// TwinCAT 3 PLC project BaseElementsSample
// ProgramVersion: 3.1.4020.1
// libraries:
//   Base_Elements,0.0.1.68,Vistaprint
//   Base_PLC,0.3.6.2,Vistaprint
//   Tc2_EtherCAT,3.3.7.0,Beckhoff Automation GmbH
//   Tc2_SerialCom,3.3.5.0,Beckhoff Automation GmbH
//   Tc2_Standard,3.3.1.0,Beckhoff Automation GmbH
//   Tc2_System,3.4.13.0,Beckhoff Automation GmbH
//   Tc2_TcpIp,3.3.3.0,Beckhoff Automation GmbH
//   Tc2_Utilities,3.3.14.0,Beckhoff Automation GmbH
//   Tc3_Interfaces,3.4.2.0,Beckhoff Automation GmbH
//   Tc3_MemMan,3.3.1.0,Beckhoff Automation GmbH
//   Tc3_Module,3.3.11.0,Beckhoff Automation GmbH
// project tree:
//   DUTs/ E_CtrlId.TcDUT, T_HashInfo.TcDUT (not stored)
//   DUTs/GVLs/ Global.TcGVL, Io.TcGVL
//   POUs/Program/ MiddlePRG_1.TcPOU, SlowPRG_1.TcPOU (not stored), FastPRG_1.TcPOU
//   / Task_Fast.TcTTO, Task_Middle.TcTTO (not stored), Task_Slow.TcTTO (not stored)
// (motion and I/O tree: see PLC project base_elements)
// real-time tasks:
//   TASK Task_Fast: cycle T#2ms, priority 4, ADS port 350
//   TASK Task_Slow: cycle T#50000us, priority 8, ADS port 351
//   TASK Task_Middle: cycle T#10ms, priority 6, ADS port 352

CONFIGURATION BaseElementsSample
    RESOURCE PLC ON TwinCAT3
        TASK Task_Fast(INTERVAL := T#2ms, PRIORITY := 4);
        PROGRAM FastPRG_1 WITH Task_Fast : FastPRG_1;
    END_RESOURCE
END_CONFIGURATION

// ---- DUTs/E_CtrlId.TcDUT
TYPE E_CtrlId :
(
	//not defined after startup...
	NONE,
	RFW_11,
	CYL_1,
	VPC_1,	
	UMC_1,	
	PRS_1,	
	BCC_1,
	DRV_1,
	RFW_12,
	ACL_1,
	VLV_1,
	ECD_1,
	E_CtrlIdMax
);
END_TYPE

// ---- DUTs/GVLs/Global.TcGVL
VAR_GLOBAL
	/// instance array of all controller instances
	g_a_pCtrlInst: ARRAY[0..E_CtrlId.E_CtrlIdMax] OF POINTER TO fb_CtrlBase;
	/// common interface array of all controllers (main use for PLC)
	g_a_pCtrlCIf: ARRAY[0..E_CtrlId.E_CtrlIdMax] OF POINTER TO T_Ctrl_CIf;
	
	/// global alarm manager
	g_p_fbAlm_Man: POINTER TO FB_Alm_Man;
	
	///Global accesss of driver init in faster cycles
	g_pFB_RFR: POINTER TO FB_RFR;	
	g_pFB_BCD: POINTER TO FB_BCD;
	g_pFB_RFD: POINTER TO FB_RFD;
	
	g_uinStartProzess : UINT; // For StartUp order
  	
END_VAR

VAR_GLOBAL CONSTANT
	c_uinCntTaskClass : UINT := 3;	// Count of Task Classes
END_VAR

// ---- DUTs/GVLs/Io.TcGVL
VAR_GLOBAL
	In_bol_11_0_B1_Doublestopper_full AT %I* : BOOL; //VOLLMELDUNG DOPPELSTOPPER
	Out_bol_11_0_Q2_Doublestopper AT %Q* : BOOL; //DOPPELSTOPPER
	In_bol_11_0_B3_Doublestopper_full AT %I* : BOOL; //VOLLMELDUNG DOPPELSTOPPER
	Out_bol_11_0_Q4_Doublestopper AT %Q* : BOOL; //DOPPELSTOPPER
	In_bol_11_0_B5_Seperator_full AT %I* : BOOL; //VOLLMELDUNG VEREINZELUNG
	In_bol_11_0_B6_Hanger_in_Seperator AT %I* : BOOL; //BUEGEL IN VEREINZELUNG
	Out_bol_11_0_Q7_Seperator AT %Q* : BOOL; //VEREINZELUNG
	Out_bol_11_0_Q8_Control_stopper AT %Q* : BOOL; //KONTROLLSTOPPER
	Out_bol_11_0_A1_Drive_On AT %Q* : BOOL; //ANTRIEB EIN
	In_bol_11_0_A1_Motor_Protection AT %I* : BOOL; //MOTORSCHUTZ AUSGELOEST
	In_bol_11_0_B13_Doublestopper_full AT %I* : BOOL; //VOLLMELDUNG DOPPELSTOPPER
	Out_bol_11_0_Q14_Doublestopper AT %Q* : BOOL; //DOPPELSTOPPER
	In_bol_11_0_B15_New_part AT %I* : BOOL; //NEUES TEIL
	In_bol_EmergencyOff AT %I* : BOOL; // Emergency Off Button
	Out_bolLED_RD AT %Q* : BOOL; // Red LED
	Out_bolLED_YE AT %Q* : BOOL; // Yellow LED
	Out_bolLED_GN AT %Q* : BOOL; // Green LED
	Out_bolBeep AT %Q* : BOOL; // Beeper
END_VAR

// ---- POUs/Program/FastPRG_1.TcPOU
PROGRAM FastPRG_1
VAR
	bolPlcStartupDone: BOOL := FALSE;
	bolHostInitDone: BOOL := FALSE;
	bolInitDone: BOOL := FALSE;

	// RFID driver
	fbRFR_11: FB_RFR;
	fbRFD_12: FB_RFD;
	// Barcode driver
	fbBCD_1: FB_BCD;
	
	fbHashTable : FB_GHT;
	uliBarcodeIn	: ULINT := 0;
	uliBarcodeOut	: ULINT := 0;

	rHashInfo	: T_HashInfo;
	pHashInfo	: POINTER TO T_HashInfo;	

END_VAR

(*__________________________________________________________________________________________________
¦	
¦	Vistaprint Schweiz GmbH
¦	CH - 8401 Winterthur
¦
¦	www.vistaprint.ch - info@vistaprint.ch
¦___________________________________________________________________________________________________

Function desription:
call of all controller (FUB) for the fast task class.

for the RFID is necessary to call to driver FUB at about 2-3ms for reaching baudhrate!

History:
Version		Date			Author		Comment
---------------------------------------------------------------------------------------------------
0.00.1		25.09.2013		AVME/KVO	Start history
0.00.2		07.01.2014		AVME/DSC 	Insert barcode driver example
0.00.3		06.01.2014		AVME/PRE	Implement RFW for Promo RFID Reader-Writer
0.00.4		13.01.2014		AVME/PRE	Implement Starup Cycle
___________________________________________________________________________________________________*)

// -----------------------------------------------------------------------------------------------
// Initialize the PLC Parameter and check the PLC health
// -----------------------------------------------------------------------------------------------
IF (NOT bolPlcStartupDone) THEN
	bolPlcStartupDone := TRUE;	
	
	// init	
	g_pFB_RFR := ADR(fbRFR_11);
	g_pFB_RFD := ADR(fbRFD_12);

	g_pFB_BCD := ADR(fbBCD_1);
	g_uinStartProzess:=1; // For StartUp order

	fbHashTable.Initialize();
END_IF
// -----------------------------------------------------------------------------------------------


// -----------------------------------------------------------------------------------------------
// The host system is downloading all parameter at startup. 
// bolPlcStartupDone will be set to true after the Host is done with the initialization
// -----------------------------------------------------------------------------------------------
IF (bolPlcStartupDone AND (NOT bolHostInitDone) AND NOT bolInitDone AND (g_uinStartProzess>=c_uinCntTaskClass)) THEN
	bolHostInitDone := TRUE;
	g_uinStartProzess := 11; // For StartUp order
END_IF
// -----------------------------------------------------------------------------------------------


// -----------------------------------------------------------------------------------------------
// Start PLC code initialization
// -----------------------------------------------------------------------------------------------
IF NOT bolInitDone AND bolPlcStartupDone AND bolHostInitDone AND (g_uinStartProzess>=(10+c_uinCntTaskClass)) THEN
		
	bolInitDone := TRUE;
	g_uinStartProzess := 21; // For StartUp order
END_IF
// -----------------------------------------------------------------------------------------------

// -----------------------------------------------------------------------------------------------
// Normal Run mode after all the initialization is done
// -----------------------------------------------------------------------------------------------
IF (bolInitDone AND bolPlcStartupDone AND bolHostInitDone AND (g_uinStartProzess>=(20+c_uinCntTaskClass))) THEN
	
	//****************************************************************************************************
	// cyclic controller calls
	//****************************************************************************************************
	//fbRFR_11();
	//fbRFD_12();
	fbBCD_1();
	
	IF uliBarcodeIn <> 0 THEN
		pHashInfo := __NEW(T_HashInfo);
		pHashInfo^.strBarcode := ULINT_TO_STRING(uliBarcodeIn);
		fbHashTable.AddItem(uliBarcodeIn, pHashInfo);
		uliBarcodeIn := 0;
	END_IF
	
	IF uliBarcodeOut <> 0 THEN
		pHashInfo := fbHashTable.Lookup(uliBarcodeOut, TRUE);
		MEMCPY(ADR(rHashInfo), pHashInfo, SIZEOF(T_HashInfo));
		__DELETE(pHashInfo);
		uliBarcodeOut := 0;
	END_IF
END_IF
// -----------------------------------------------------------------------------------------------

END_PROGRAM

// ---- POUs/Program/MiddlePRG_1.TcPOU
PROGRAM MiddlePRG_1
VAR
	fbAlm_Man: FB_Alm_Man; // alarm manager
	
	bolPlcStartupDone: BOOL := FALSE;
	bolHostInitDone: BOOL := FALSE;
	bolInitDone: BOOL := FALSE;
	uinTaskNbr : UINT := 2; // MiddleTask is Task Nr 2
	fbRFW_11: FB_RFW;
	fbRFW_12: FB_RFW;
	fbBCC_1: FB_BCC;
	fbCYL_1: FB_CYL;
	fbPRS_1: FB_PRS;
	fbUMC_1: FB_UMC;
	fbVPC_1: FB_VPC;
	fbDRV_1: FB_DRV;
	pTmpSIf_RFW: POINTER TO Base_Elements.T_Ctrl_SIf_RFW;
	pTmpSIf_BCC: POINTER TO T_Ctrl_SIf_BCC;
	fbVLV_1: FB_VLV;
	
	// ADS Client Example
	fbACL_1: FB_ACL;
	sCon01_ShirtStream: T_ADS_ConnectionData; 			// Example: Read connection to shirt stream PLC (Port 851) drive FUB interface .cur
	DrvCurData: T_Ctrl_SIf_DRV_Cur;	
	sCon02_ShirtStream: T_ADS_ConnectionData; 			// Example: Write connection to shirt stream PLC (Port 851) drive FUB interface .par
	DrvParData: T_Ctrl_SIf_DRV_Par;	
	sCon03_ShirtStream: T_ADS_ConnectionData; 			// Example: Write connection to shirt stream PLC (Port 852) drive FUB interface .cfg
	DrvCfgData: T_Ctrl_SIf_DRV_Cfg;	
	// ADS Client Example
	
	// EtherCAT Diagnose
	fbECD_1: FB_ECD;
	pTmpSIf_ECD: POINTER TO T_Ctrl_SIf_ECD;

	fbSGT_1: 		FB_SGT;		// Signal tower	
	pDRV_CIf:		POINTER TO Base_PLC.T_Ctrl_CIf; // Used for Signal tower example
	pDRV_SIf:		POINTER TO Base_Elements.T_Ctrl_SIf_DRV; // Used for Signal tower example
	
	// close all Ethernet sockets
	fbSocketCloseAll : FB_SocketCloseAll;
END_VAR

(*__________________________________________________________________________________________________
¦	
¦	Vistaprint Schweiz GmbH
¦	CH - 8401 Winterthur
¦
¦	www.vistaprint.ch - info@vistaprint.ch
¦___________________________________________________________________________________________________

Function desription:
call of all controller (FUB) for the middle task class.


History:
Version		Date			Author		Comment
---------------------------------------------------------------------------------------------------
0.00.1		25.09.2013		AVME/KVO	Start history
0.00.2		12.11.2013		VP/RE		Local AlarmManager
0.00.3		07.01.2014		AVME/DSC 	Insert barcode reader example
0.00.4		08.01.2014		AVME/MRU	Insert DRV example
0.00.5		06.01.2014		AVME/PRE	Implement RFW for Promo Read and Write RFID Reader
0.00.6		13.01.2014		AVME/PRE	Implement Starting Up Process
0.00.7		05.02.2014		AVME/DSC	Insert ADS client example
0.00.8		06.03.2014		AVME/DSC	Insert FB_VLV example
0.00.9		17.06.2014		AVME/MRU	SGT example added
0.00.10		24.10.2014		HLV/MAH		close all sockets on PLC init

___________________________________________________________________________________________________*)

// -----------------------------------------------------------------------------------------------
// Initialize the PLC Parameter and check the PLC health
// -----------------------------------------------------------------------------------------------
IF (NOT bolPlcStartupDone) AND (g_uinStartProzess>=(uinTaskNbr-1)) THEN
	
	// init	
	// Level0 -------------------------------------------------------------------
	
	// RFID Reader, element Controller in this Task, Driver in fastest Task class
	fbRFW_11.iniAllCtrlArrays(ADR(g_a_pCtrlInst),ADR(g_a_pCtrlCIf),E_CtrlId.RFW_11); // init and entry fb_instance in global fb pointer array
	fbRFW_11.pRFD_SIf := g_pFB_RFR^.getSIf();
	pTmpSIf_RFW := fbRFW_11.getCtrlSIf();
	pTmpSIf_RFW^.Cfg.eTyp := E_Typ_RFW.RF382R;
	// the following parameters are not needed at the moment because the parameters will not be written down for RF382R at the moment
	pTmpSIf_RFW^.Cfg.stNetId := '192.168.2.123.1.1'; //PLC NetId
	pTmpSIf_RFW^.Cfg.uinSlaveAddr := 1024; //Io card Ethercat adress 
	pTmpSIf_RFW^.Cfg.bolGetTrayIDAuto := FALSE;
	
	// RFID Reader, element Controller in this Task, Drive in fastest Task class
	fbRFW_12.iniAllCtrlArrays(ADR(g_a_pCtrlInst),ADR(g_a_pCtrlCIf),E_CtrlId.RFW_12); // init and entry fb_instance in global fb pointer array
	fbRFW_12.pRFD_SIf := g_pFB_RFD^.getSIf();
	pTmpSIf_RFW := fbRFW_12.getCtrlSIf();
	pTmpSIf_RFW^.Cfg.eTyp := E_Typ_RFW.RF310R;
	// the following parameters are not needed at the moment because the parameters will not be written down for RF382R at the moment
	pTmpSIf_RFW^.Cfg.stNetId := '192.168.2.123.1.1'; //PLC NetId
	pTmpSIf_RFW^.Cfg.uinSlaveAddr := 1024; //Io card Ethercat adress 
	pTmpSIf_RFW^.Cfg.bolGetTrayIDAuto := TRUE;
	
	// *********************************************************
	// Barcode reader example
	// *********************************************************
	
	// Barcode reader, element Controller in this Task, Driver in fastest Task class
	fbBCC_1.iniAllCtrlArrays(ADR(g_a_pCtrlInst),ADR(g_a_pCtrlCIf),E_CtrlId.BCC_1); // init and entry fb_instance in global fb pointer array
	fbBCC_1.pBCD_SIf_In := g_pFB_BCD^.getSIf();
	pTmpSIf_BCC := fbBCC_1.getCtrlSIf();
	// configuration	
	pTmpSIf_BCC^.Cfg.strSensorIPAdr := '192.168.70.28';
	pTmpSIf_BCC^.Cfg.udiSensorPort := 2111;
	pTmpSIf_BCC^.Cfg.iSensorType := E_BCD_Type.SICK;
	(*
	pTmpSIf_BCC^.Cfg.strSensorIPAdr := '192.168.1.103';
	pTmpSIf_BCC^.Cfg.udiSensorPort := 9004;
	pTmpSIf_BCC^.Cfg.iSensorType := E_BCD_Type.KEYENCE;
	*)
	// *********************************************************
	// ADS client example
	// *********************************************************
	
	// ADS client connection
	fbACL_1.iniAllCtrlArrays(ADR(g_a_pCtrlInst),ADR(g_a_pCtrlCIf),E_CtrlId.ACL_1); // init and entry fb_instance in global fb pointer array

	// Add a read connection
	sCon01_ShirtStream.eAccessType := E_ADS_AccessType.READ;
	sCon01_ShirtStream.uinTargetPort:= 851;
	sCon01_ShirtStream.strNetID := '192.168.70.27.1.1';
	sCon01_ShirtStream.strRoute := 'SlowPRG_1.fbDRV_1.SIf.Cur';
	sCon01_ShirtStream.udiDataLen:= SIZEOF(DrvCurData);
	sCon01_ShirtStream.pData:= ADR(DrvCurData);	
	// Add defined connection to client
	fbACL_1.AddConnection(sCon01_ShirtStream);

	// Add a write connection
	sCon02_ShirtStream.eAccessType := E_ADS_AccessType.WRITE;
	sCon02_ShirtStream.uinTargetPort:= 851;
	sCon02_ShirtStream.strNetID := '192.168.70.27.1.1';
	sCon02_ShirtStream.strRoute := 'SlowPRG_1.fbDRV_1.SIf.Par';
	sCon02_ShirtStream.udiDataLen:= SIZEOF(DrvParData);
	sCon02_ShirtStream.pData:= ADR(DrvParData);	
	// Add defined connection to client
	fbACL_1.AddConnection(sCon02_ShirtStream);
	
	// Add a write connection
	sCon03_ShirtStream.eAccessType := E_ADS_AccessType.WRITE;
	sCon03_ShirtStream.uinTargetPort:= 852;
	sCon03_ShirtStream.strNetID := '192.168.70.27.1.1';
	sCon03_ShirtStream.strRoute := 'SlowPRG_1.fbDRV_1.SIf.Cfg';
	sCon03_ShirtStream.udiDataLen:= SIZEOF(DrvCfgData);
	sCon03_ShirtStream.pData:= ADR(DrvCfgData);	
	// Add defined connection to client
	fbACL_1.AddConnection(sCon03_ShirtStream);
	
	// More connections can be insert here ... !
	
	
	
	// *********************************************************
	// Different controller
	// *********************************************************
	
	// cylinder example
	fbCYL_1.iniAllCtrlArrays(ADR(g_a_pCtrlInst),ADR(g_a_pCtrlCIf),E_CtrlId.CYL_1); // init and entry fb_instance in global fb pointer array
	fbPRS_1.iniAllCtrlArrays(ADR(g_a_pCtrlInst),ADR(g_a_pCtrlCIf),E_CtrlId.PRS_1); // init and entry fb_instance in global fb pointer array
	fbUMC_1.iniAllCtrlArrays(ADR(g_a_pCtrlInst),ADR(g_a_pCtrlCIf),E_CtrlId.UMC_1); // init and entry fb_instance in global fb pointer array
	fbVPC_1.iniAllCtrlArrays(ADR(g_a_pCtrlInst),ADR(g_a_pCtrlCIf),E_CtrlId.VPC_1); // init and entry fb_instance in global fb pointer array
	fbDRV_1.iniAllCtrlArrays(ADR(g_a_pCtrlInst),ADR(g_a_pCtrlCIf),E_CtrlId.DRV_1); // init and entry fb_instance in global fb pointer array
	fbVLV_1.iniAllCtrlArrays(ADR(g_a_pCtrlInst),ADR(g_a_pCtrlCIf),E_CtrlId.VLV_1); // init and entry fb_instance in global fb pointer array	
	
	// set command to close all socket connections
	fbSocketCloseAll.bExecute := TRUE;
	
	bolPlcStartupDone := TRUE;	
	g_uinStartProzess := g_uinStartProzess + 1; // For StartUp order
	
		// EtherCAT Diagnostic Element
	fbECD_1.iniAllCtrlArrays(ADR(g_a_pCtrlInst),ADR(g_a_pCtrlCIf),E_CtrlId.ECD_1); // init and entry fb_instance in global fb pointer array
	pTmpSIf_ECD := fbECD_1.getCtrlSIf();
	pTmpSIf_ECD^.Cfg.strNetID := '192.168.70.24.2.1'; //PLC NetId

END_IF
// -----------------------------------------------------------------------------------------------


// -----------------------------------------------------------------------------------------------
// The host system is downloading all parameter at startup. 
// bolPlcStartupDone will be set to true after the Host is done with the initialization
// -----------------------------------------------------------------------------------------------
IF (bolPlcStartupDone AND (NOT bolHostInitDone) AND NOT bolInitDone AND (g_uinStartProzess>=(uinTaskNbr-1)+10)) THEN
	bolHostInitDone := TRUE;
	g_uinStartProzess := g_uinStartProzess + 1; // For StartUp order
END_IF
// -----------------------------------------------------------------------------------------------


// -----------------------------------------------------------------------------------------------
// Start PLC code initialization
// -----------------------------------------------------------------------------------------------
IF NOT bolInitDone AND bolPlcStartupDone AND bolHostInitDone AND (g_uinStartProzess>=(uinTaskNbr-1)+20) THEN
	
	// call FB to close all socket connections
	fbSocketCloseAll();
	fbSocketCloseAll.bExecute := FALSE;

	IF fbSocketCloseAll.bBusy = FALSE THEN
		bolInitDone := TRUE;
	END_IF
	g_uinStartProzess := g_uinStartProzess + 1; // For StartUp order
END_IF
// -----------------------------------------------------------------------------------------------

// -----------------------------------------------------------------------------------------------
// Normal Run mode after all the initialization is done
// -----------------------------------------------------------------------------------------------
IF (bolInitDone AND bolPlcStartupDone AND bolHostInitDone AND (g_uinStartProzess>=(20+c_uinCntTaskClass))) THEN
	
	//****************************************************************************************************
	// cyclic controller calls
	//****************************************************************************************************
	fbRFW_11();
	fbRFW_12();
	fbCYL_1();
	fbPRS_1();
	fbUMC_1();
	fbVPC_1();
	fbDRV_1();
	fbVLV_1();
	
	fbBCC_1();   // Barcode reader example
	fbACL_1();		// ADS client example
		
	fbECD_1(); // EtherCAT Diagnostic
	
	// --------------------------------------------------
	// Signal tower
	// --------------------------------------------------

	// Signal tower conditions for red, yellow and green
	// -------------------------------------------------
	
	// Get access to FB_DRV
	pDRV_CIf := fbDRV_1.CtrlCIf;
	pDRV_SIf := fbDRV_1.getCtrlSIf();
	
	// GreenBlink
	IF (pDRV_CIf^.Job.intState = Base_PLC.cSTA_RUNBusy) THEN
		fbSGT_1.In_bolGreenBlink:= TRUE;
	ELSE
		fbSGT_1.In_bolGreenBlink:= FALSE;
	END_IF
	
	// GreenOn
	IF (pDRV_CIf^.Job.intState = Base_PLC.cSTA_RUN) THEN
		fbSGT_1.In_bolGreenOn:= TRUE;
	ELSE
		fbSGT_1.In_bolGreenOn:= FALSE;
	END_IF
	
(*	// Yellow
	fbSGT_1.In_uinCntYellow:= pDRV_SIf^.Cur.uinNrOfActiveInfo;
	// Red
	fbSGT_1.In_uinCntRed:= pDRV_SIf^.Cur.uinNrOfActiveAlarm;
	// Beep (only in case of an alarm)
	fbSGT_1.In_uinCntBeep:= pDRV_SIf^.Cur.uinNrOfActiveAlarm;
*)
	// Call SGT 
	fbSGT_1();	
	Out_bolLED_RD:= fbSGT_1.Out_bolRed;
	Out_bolLED_YE:= fbSGT_1.Out_bolYellow;
	Out_bolLED_GN:= fbSGT_1.Out_bolGreen;	
	Out_bolBeep:= fbSGT_1.Out_bolBeep;
	
END_IF
// -----------------------------------------------------------------------------------------------

END_PROGRAM
